RoboDK station: Proyecto_Grupo3_P105.rdk

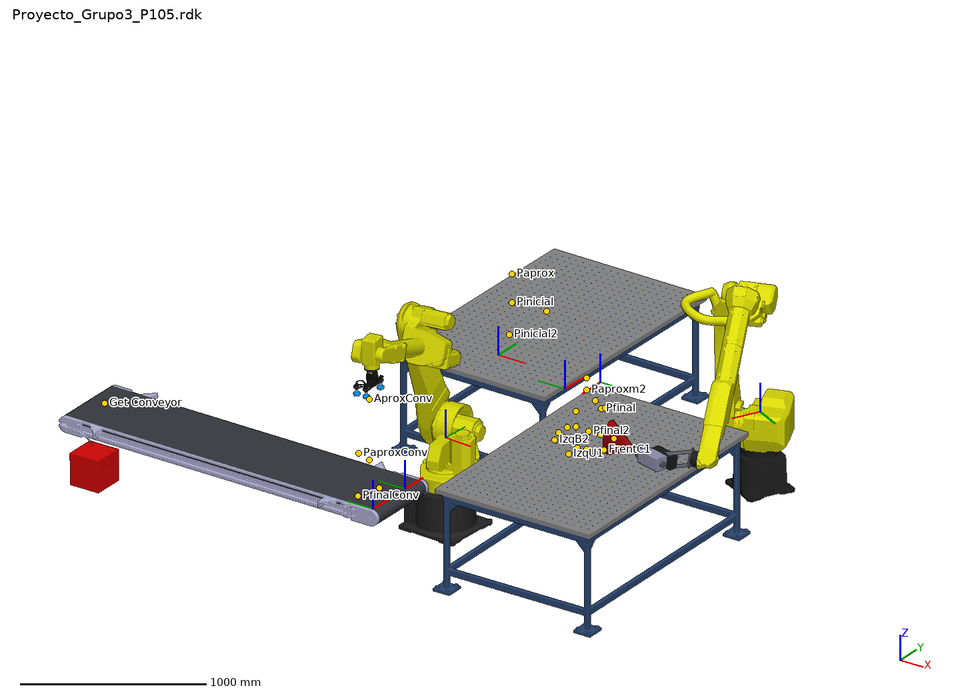
[picture v0: the station drawn from its stored meshes, robots at their saved joint values, targets as dots, program paths as lines]
Station ProyectoConConv (saved by RoboDK 5.3.0). Poses are relative to the parent item; angles as X-Y-Z fixed-axis rotations.
Station parameters (name, value as stored): ColorCilindro, 3.0
  - frame Fanuc M-16iB/20 Base at (-465.89, -504.82, 525) mm, rotated rx 0 ry 0 rz -2.81 deg
    - robot Fanuc M-16iB/20: 6 axes, payload 20 kg, reach 1667 mm, repeatability 0.08 mm, weight 270 kg
        modified DH rows (alpha deg, a mm, theta deg, d mm): 0, 0, 0, 525; -90, 150, -90, 0; 0, 770, 0, 0; -90, 100, 0, 740; 90, 0, 0, 0; -90, 0, 0, 100
        base shift (0, 0, -525) mm
        joint limits [-170, -90, -170, -200, -140, -450] to [170, 160, 290, 200, 140, 450]; home [0, 0, 0, 0, -90, 0]; saved at [100.119, -20.895, 160.194, 178.685, -110.161, -367.731]
      - tool RobotiQ EPick Four Vacuum Cup, TCP at (0, 21.99, 131.95) mm, size 175.2 x 107.7 x 135.6 mm
    - target Pfinal (Cartesian target) at (967.03, 121.53, 415.61) mm, rotated rx -178.82 ry 0.51 rz 89.06 deg; joints [7.493, 4.996, -18.964, 0.352, -72.278, -278.545] of Fanuc M-16iB/20
    - target PfinalConv (Cartesian target) at (196.13, -1019.55, 104.82) mm, rotated rx -178.83 ry 0.51 rz 177.59 deg; joints [-79.527, 21.76, -40.518, -0.315, -48.231, -102.682] of Fanuc M-16iB/20
    - target PaproxConv (Cartesian target) at (194.18, -1012.63, 357.54) mm, rotated rx -178.83 ry 0.51 rz 177.59 deg; joints [-79.563, 13.7, -22.039, -0.256, -66.709, -102.754] of Fanuc M-16iB/20
    - frame Est1 at (-300.91, 850, 79.96) mm, rotated rx 0 ry 0 rz 2.81 deg
      - target Paprox (Cartesian target) at (92.49, 0.53, 509.87) mm, rotated rx -178.82 ry 0.51 rz 89.06 deg; joints [105.312, -0.649, -5.743, 178.728, 84.484, -193.315] of Fanuc M-16iB/20
      - target Pinicial2 (Cartesian target) at (75, 0, 140) mm, rotated rx -180 ry 0.52 rz 90 deg; joints [-73.822, -24.597, 187.698, -180.122, -82.809, -13.348] of Fanuc M-16iB/20
      - target Pinicial (Cartesian target) at (93.45, -1.01, 339.4) mm, rotated rx -178.82 ry 0.51 rz 89.06 deg; joints [105.273, 0.25, -18.897, -1.336, -71.334, -372.97] of Fanuc M-16iB/20
      - target P2Inicial (Cartesian target) at (75, 350, 140) mm, rotated rx -178.82 ry 0.51 rz 90 deg; joints [102.152, 27.689, -21.607, -1.338, -68.714, -368.854] of Fanuc M-16iB/20
    - frame Est2 at (346.71, 909.84, 87.05) mm, rotated rx 0 ry 0 rz -86.3 deg
      - object Estacion2 at (1300, 499.97, 0) mm, rotated rx 0 ry 0 rz -180 deg, size 1535.8 x 1018.8 x 608.3 mm, geometry from Table-2000mmx1200mmx800mm.sld
      - target Paproxm2 (Cartesian target) at (800, 455.71, 400) mm, rotated rx 180 ry 0 rz 90 deg; joints [11.351, -2.011, -4.047, 0, -85.953, -367.648] of Fanuc M-16iB/20
      - target Pfinal2 (Cartesian target) at (775, 450, 140) mm, rotated rx -180 ry 0 rz 0 deg; joints [10.89, 2.514, -28.094, 0, -61.906, -97.187] of Fanuc M-16iB/20
      - object Estacion1 at (17.89, -650.14, -7.09) mm, rotated rx 0 ry 0 rz 179.11 deg, size 1535.8 x 1018.8 x 608.3 mm, geometry from Table-2000mmx1200mmx800mm.sld
  - Python program Set (listed below)
  - Python program Prepare (listed below)
  - Python program Robot1_2 (listed below)
  - Python program Robot2_Conv (listed below)
  - Python program Robot2_2 (listed below)
  - Python program SensorActivate (listed below)
  - frame Fanuc M-10iA/8L Base at (643.98, 857.38, 450) mm, rotated rx 0 ry 0 rz -116.36 deg
    - robot Fanuc M-10iA/8L: 6 axes, payload 8 kg, reach 2028 mm, repeatability 0.04 mm, weight 150 kg
        modified DH rows (alpha deg, a mm, theta deg, d mm): 0, 0, 0, 450; -90, 150, -90, 0; 0, 780, 0, 0; -90, 200, 0, 1080; 90, 0, 0, 0; -90, 0, 0, 100
        base shift (0, 0, -450) mm
        joint limits [-170, -90, -180, -200, -140, -270] to [170, 160, 267, 200, 140, 270]; home [12.06, 4.62, 10.35, -4.26, -75.46, -178.09]; saved at [47.67, 3.001, -39.586, 91.935, -94.481, -221.235]
      - tool Paint gun, TCP at (50, 0, 450) mm, rotated rx 0 ry 30 rz 0 deg, size 203.2 x 279.7 x 471.5 mm
    - target AproxPin (Cartesian target) at (1241.53, 330.16, 632.23) mm, rotated rx -179.35 ry -2.45 rz -157.72 deg; joints [13.753, -7.97, 9.222, -3.553, -71.889, -170.998] of Fanuc M-10iA/8L
    - target IzqU1 (Cartesian target) at (1385.42, 391.79, 236.72) mm, rotated rx 175.16 ry -45.65 rz -162.72 deg; joints [14.487, 30.06, -6.496, -3.483, -99.223, -180.287] of Fanuc M-10iA/8L
    - target IzqU2 (Cartesian target) at (1386.34, 378.43, 391.89) mm, rotated rx -176.7 ry -51.36 rz -166.63 deg; joints [15.972, 36.806, 3.248, 2.102, -114.653, -179.895] of Fanuc M-10iA/8L
    - target Sup1 (Cartesian target) at (1323.33, 361.68, 464.26) mm, rotated rx -179.35 ry -2.45 rz -157.72 deg; joints [14.303, -4.968, -0.111, -3.521, -62.54, -170.968] of Fanuc M-10iA/8L
    - target Sup2 (Cartesian target) at (1176.85, 310.11, 472.26) mm, rotated rx -178 ry 0.46 rz -156.27 deg; joints [13.626, -18.1, 1.596, -3.869, -61.306, -168.43] of Fanuc M-10iA/8L
    - target DerU1 (Cartesian target) at (1096.06, 271.61, 393.16) mm, rotated rx -177.41 ry 39.38 rz -154.65 deg; joints [7.092, -50.059, -3.563, -40.967, -22.985, -133.522] of Fanuc M-10iA/8L
    - target DerU2 (Cartesian target) at (1129.24, 280.47, 243.27) mm, rotated rx -176.98 ry 48.64 rz -154.02 deg; joints [6.444, -49.98, -15.791, -103.175, -16.992, -70.804] of Fanuc M-10iA/8L
    - target IzqB1 (Cartesian target) at (1352.99, 430.79, 281.25) mm, rotated rx 98.01 ry -2.72 rz -102.48 deg; joints [3.224, 45.691, -20.072, -62.199, -126.893, -145.453] of Fanuc M-10iA/8L
    - target IzqB2 (Cartesian target) at (1432.32, 316.89, 300.11) mm, rotated rx 98.01 ry -2.72 rz -102.48 deg; joints [-0.403, 53.002, -15.112, -63.442, -132.237, -149.123] of Fanuc M-10iA/8L
    - target AtrasB1 (Cartesian target) at (1371.24, 253.12, 300.21) mm, rotated rx 98.01 ry -2.72 rz -102.48 deg; joints [-2.438, 46.986, -18.398, -59.38, -132.376, -143.961] of Fanuc M-10iA/8L
    - target AtrasB2 (Cartesian target) at (1241.59, 206.8, 287.27) mm, rotated rx 98.01 ry -2.72 rz -102.48 deg; joints [-4.203, 36.509, -24.123, -53.707, -130.589, -136.372] of Fanuc M-10iA/8L
    - target IzqC1 (Cartesian target) at (1377.37, 326.06, 306.96) mm, rotated rx -88.88 ry 4.57 rz 171.9 deg; joints [-144.988, -47.039, 182.818, -87.325, -103.378, 174.474] of Fanuc M-10iA/8L
    - target IzqC2 (Cartesian target) at (1332.28, 498.61, 298.22) mm, rotated rx -90.14 ry 4.7 rz 156.34 deg; joints [-141.526, -71.736, 167.629, -79.805, -120.795, 191.683] of Fanuc M-10iA/8L
    - target FrentC1 (Cartesian target) at (1247.52, 535.75, 290.61) mm, rotated rx -87.43 ry 3.94 rz -168.8 deg; joints [-133.276, -36.716, 189.36, -86.769, -96.288, 168.888] of Fanuc M-10iA/8L
    - target FrentC2 (Cartesian target) at (1130.62, 430.13, 284.93) mm, rotated rx -87.14 ry 3.73 rz -164.4 deg; joints [-132.33, -23.306, 194.93, -86.372, -93.265, 163.449] of Fanuc M-10iA/8L
  - Python program pintura (listed below)
  - Python program SprayOn (listed below)
  - program MainProgram (15 instructions, listed below)
  - Python program Prog12 (listed below)
  - Python program PinturaP2 (listed below)
  - frame ConveyorReference at (-173.28, -1600, 618.68) mm, rotated rx 0 ry 0 rz 90.03 deg
    - target Get Conveyor (Cartesian target) at (200, 1900, 20) mm, rotated rx 90 ry 0 rz 0 deg; joints [0, 0, 0, 0, 0, 43.699]
    - frame Final_conv at (1800, 0, 0) mm
    - target Put Conveyor (Cartesian target) at (200, 100, 20) mm, rotated rx 90 ry 0 rz -180 deg; joints [134.006, 22.86, -66.558, 43.699, -45.994, 0]
    - object Conveyor at (0, 300, -50) mm, size 597 x 2090.8 x 107.2 mm
      - Python program RunConveyor (listed below)
      - Python program WaitForPart (listed below)
      - Python program SimulateGripper (listed below)
      - object box at (316.14, 335.9, 144.87) mm, rotated rx 0.06 ry -0.07 rz 75.08 deg, size 125 x 125 x 125 mm, geometry from box.sld
      - object Part 1 at (249.98, 1701.74, -449.97) mm, rotated rx 0.01 ry 1.18 rz 89.99 deg, size 187.5 x 187.5 x 187.5 mm, geometry from box.sld
      - object Part 2 at (250, 1704, -450) mm, rotated rx 0 ry 0 rz 90 deg, size 187.5 x 187.5 x 187.5 mm, geometry from box.sld
    - frame Inicial_conv at (300, 0, 0) mm
    - target FinalConv (Cartesian target) at (250, 200, 140) mm, rotated rx -178.82 ry 0.51 rz -180 deg; joints [100.119, -21.731, 187.781, 178.755, -82.581, -367.117] of Fanuc M-16iB/20
    - target AproxConv (Cartesian target) at (250, 200, 500) mm, rotated rx -178.82 ry 0.51 rz -180 deg; joints [100.119, -20.895, 160.194, 178.685, -110.161, -367.731] of Fanuc M-16iB/20

--- Python program Set ---
# Type help("robolink") or help("robodk") for more information
# Press F5 to run the script
# Note: you do not need to keep a copy of this file, your python script is saved with the station
from robolink import *    # API to communicate with RoboDK
from robodk import *      # basic matrix operations


#PARAM_SIZE_BOX = 'SizeBox'
#PARAM_SIZE_PALLET = 'SizePallet'
#PARAM_CONV_SPEED_MM = 'ConvSpeed'
PARAM_COLOR= 'ColorCilindro'



RDK = Robolink()

#size_box = RDK.getParam(PARAM_SIZE_BOX)
#size_pallet = RDK.getParam(PARAM_SIZE_PALLET)
#conv_speed = RDK.getParam(PARAM_CONV_SPEED_MM)
color = RDK.getParam(PARAM_COLOR)

# ------------------------------------------------------------
#size_box_input = mbox('Enter the size of the box in mm [L,W,H]', entry=size_box)
#if size_box_input:
#    RDK.setParam(PARAM_SIZE_BOX, size_box_input)
#else:
#    raise Exception('Operation cancelled by user')

# ------------------------------------------------------------
#size_pallet_input = mbox('Enter the size of the pallet', entry=size_pallet)
#if size_pallet_input:
#    RDK.setParam(PARAM_SIZE_PALLET, size_pallet_input)
#else:
#    raise Exception('Operation cancelled by user')

# ------------------------------------------------------------
#conv_speed_input = mbox('Enter the speed of the conveyor in mm/s', entry=conv_speed)
#if conv_speed_input:
#    RDK.setParam(PARAM_CONV_SPEED_MM, conv_speed_input)
#    conv_speed = float(conv_speed_input)
#    conv = RDK.Item('Conveyor Belt', ITEM_TYPE_ROBOT)
#    conv.setSpeed(conv_speed)

#else:
#    raise Exception('Operation cancelled by user')

# ------------------------------------------------------------
color_cilindro_input = mbox('Ingrese el color: 1:Amarillo 2:Azul 3:Rojo 4:Verde', entry=color)
if color_cilindro_input:
    RDK.setParam(PARAM_COLOR, color_cilindro_input)

else:
    raise Exception('Operation cancelled by user')

--- Python program Prepare ---
# Type help("robolink") or help("robodk") for more information
# Press F5 to run the script
# Note: you do not need to keep a copy of this file, your python script is saved with the station
from robolink import *    # API to communicate with RoboDK
from robodk import *      # basic matrix operations

# Use RoboDK API as RL
RDK = Robolink()

frame_pallet        = RDK.Item('Est1', ITEM_TYPE_FRAME)

# get variable parameters
#SIZE_BOX = RDK.getParam('SizeBox')
#SIZE_PALLET = RDK.getParam('SizePallet')
SIZE_BOX = [150,150,150]
SIZE_PALLET = [1,2,1]
#SIZE_BOX_XYZ = [float(x.replace(' ','')) for x in SIZE_BOX.split(',')]
#SIZE_PALLET_XYZ = [float(x.replace(' ','')) for x in SIZE_PALLET.split(',')]
SIZE_BOX_XYZ = [150,150,150]
SIZE_PALLET_XYZ = [1,2,1]
SIZE_BOX_Z = SIZE_BOX_XYZ[2] # the height of the boxes is important to take into account when approaching the positions

#COLOR_CILINDRO = RDK.getParam('ColorCilindro')
#COLOR_CILINDRO_RGB = [float(x.replace(' ','')) for x in COLOR_CILINDRO.split(',')]

def box_calc(size_xyz, pallet_xyz):
    """Calculates a list of points to store parts in a pallet"""
    [size_x, size_y, size_z] = size_xyz
    [pallet_x, pallet_y, pallet_z] = pallet_xyz
    xyz_list = []
    for h in range(int(pallet_z)):
        for j in range(int(pallet_y)):
            for i in range(int(pallet_x)):
                xyz_list = xyz_list + [[(i+0.5)*size_x, (j)*(size_y+200), (h+0)*size_z]]
    return xyz_list

def parts_setup(frame, positions, size_xyz):
    """Place a list of parts in a reference frame. The part/reference object must have been previously copied to the clipboard."""
    [size_x, size_y, size_z] = size_xyz
    nparts = len(positions)
    cstep = 1.0/(nparts - 1)
    for i in range(nparts):
        newpart = frame.Paste()
        newpart.Scale([(size_x/100), size_y/100, size_z/100]) #scale with respect to the reference object (100mm cube)
        newpart.setName('Part ' + str(i+1)) #set item name
        newpart.setPose(transl(positions[i])) #set item position with respect to parent
        newpart.setVisible(True, False) #make item visible but hide the reference frame
        newpart.Recolor([255/255,255/255,255/255,1]) #set RGBA color
#newpart.Recolor([1-cstep*i, cstep*i, 0.4, 1]) #set RGBA color

def cleanup(objects, startswith="Part "):
    """Deletes all objects where the name starts with "startswith", from the provided list of objects."""
    for item in objects:
        if item.Name().startswith(startswith):
            item.Delete()

# turn off rendering (much faster when setting up the station)
RDK.Render(False)

# cleanup previous simulation (generated parts and tools)
all_objects = RDK.ItemList(ITEM_TYPE_OBJECT, False)
cleanup(all_objects, 'Part ')
all_tools = RDK.ItemList(ITEM_TYPE_TOOL, False)
cleanup(all_tools, 'TCP ')

# copy the reference part
partref = RDK.Item('box')
partref.Copy()

#RL.Set_Simulation_Speed(500);
#RL.Set_Simulation_Mode(1)

# calculate an array of positions to get/store the parts
parts_positions = box_calc(SIZE_BOX_XYZ, SIZE_PALLET_XYZ)

# setup/initialise the parts on the palled
parts_setup(frame_pallet, parts_positions, SIZE_BOX_XYZ)

RDK.Render(True)

--- Python program Robot1_2 ---
# Type help("robolink") or help("robodk") for more information
# Press F5 to run the script
# Note: you do not need to keep a copy of this file, your python script is saved with the station
from robolink import *    # API to communicate with RoboDK
from robodk import *      # basic matrix operations

# Use RoboDK API as RL
RDK = Robolink()

# define default approach distance
APPROACH = 100

# gather robot, tool and reference frames from the station
robot = RDK.Item('Fanuc M-16iB/20', ITEM_TYPE_ROBOT)
tool = RDK.Item('RobotiQ EPick Four Vacuum Cup', ITEM_TYPE_TOOL)
frame_pallet = RDK.Item('Est1', ITEM_TYPE_FRAME)
frame_pallet2 = RDK.Item('Est2', ITEM_TYPE_FRAME)


# gather targets
target_aprox = RDK.Item('Paprox', ITEM_TYPE_TARGET)
target_aprox2 = RDK.Item('Paproxm2', ITEM_TYPE_TARGET)
target_final = RDK.Item('Pfinal2', ITEM_TYPE_TARGET)
target_inicial = RDK.Item('Pinicial2', ITEM_TYPE_TARGET)



def TCP_On(toolitem):
    """Attaches the closest object to the toolitem Htool pose,
    It will also output appropriate function calls on the generated robot program (call to TCP_On)"""
    toolitem.AttachClosest()
    toolitem.RDK().RunMessage('Set air valve on')
    toolitem.RDK().RunProgram('TCP_On()')

def TCP_Off(toolitem, itemleave=0):
    """Detaches the closest object attached to the toolitem Htool pose,
    It will also output appropriate function calls on the generated robot program (call to TCP_Off)"""
    toolitem.DetachAll(itemleave)
    toolitem.RDK().RunMessage('Set air valve off')
    toolitem.RDK().RunProgram('TCP_Off()')



# ---------------------------------------------------------------------------------
# -------------------------- PROGRAM START ----------------------------------------

tool_xyzrpw = tool.PoseTool()*transl(0,0,50)
tool_tcp = robot.AddTool(tool_xyzrpw, 'TCP A')

robot.setPoseTool(tool_tcp)
robot.setSpeed(100)
robot.setPoseFrame(frame_pallet)
robot.MoveJ(target_aprox)
#target_i_app = target_inicial * transl(0,0,-(APPROACH+50))
#robot.MoveJ(target_i_app)
#TCP_On(tool)
robot.MoveL(target_inicial)
robot.setSpeed(100)
TCP_On(tool)
#obj.setParentStatic(tool)
#TCP_On(tool)
#robot.MoveL(target_i_app)
robot.MoveL(target_aprox)
robot.setSpeed(100)
#TCP_On(tool)
robot.setPoseFrame(frame_pallet2)
robot.MoveL(target_aprox2)
robot.setSpeed(100)
robot.MoveL(target_final)
#robot.MoveJ(target_inicial)
TCP_Off(tool, frame_pallet2)
robot.MoveJ(target_aprox2)
robot.setPoseFrame(frame_pallet)
robot.MoveL(target_aprox)


def cleanup(objects, startswith="Part "):
    """Deletes all objects where the name starts with "startswith", from the provided list of objects."""
    for item in objects:
        if item.Name().startswith(startswith):
            item.Delete()

# turn off rendering (much faster when setting up the station)
RDK.Render(False)

# cleanup previous simulation (generated parts and tools)

all_tools = RDK.ItemList(ITEM_TYPE_TOOL, False)
cleanup(all_tools, 'TCP ')

--- Python program Robot2_Conv ---
# Type help("robolink") or help("robodk") for more information
# Press F5 to run the script
# Note: you do not need to keep a copy of this file, your python script is saved with the station
from robolink import *    # API to communicate with RoboDK
from robodk import *      # basic matrix operations

# Use RoboDK API as RL
RDK = Robolink()

# define default approach distance
#APPROACH = 100

# gather robot, tool and reference frames from the station
robot = RDK.Item('Fanuc M-16iB/20', ITEM_TYPE_ROBOT)
tool = RDK.Item('RobotiQ EPick Four Vacuum Cup', ITEM_TYPE_TOOL)
#obj = RDK.Item('box', ITEM_TYPE_OBJECT)
frame_pallet = RDK.Item('Est2', ITEM_TYPE_FRAME)
frame_pallet2 = RDK.Item('ConveyorReference', ITEM_TYPE_FRAME)
#frame_conv          = RDK.Item('ConveyorReference', ITEM_TYPE_FRAME)
#frame_conv_moving   = RDK.Item('MovingRef', ITEM_TYPE_FRAME)

# gather targets
target_aprox = RDK.Item('Paproxm2', ITEM_TYPE_TARGET)
target_aprox2 = RDK.Item('AproxConv', ITEM_TYPE_TARGET)
target_final = RDK.Item('FinalConv', ITEM_TYPE_TARGET)
target_inicial = RDK.Item('Pfinal2', ITEM_TYPE_TARGET)



def TCP_On(toolitem):
    """Attaches the closest object to the toolitem Htool pose,
    It will also output appropriate function calls on the generated robot program (call to TCP_On)"""
    toolitem.AttachClosest()
    toolitem.RDK().RunMessage('Set air valve on')
    toolitem.RDK().RunProgram('TCP_On()')

def TCP_Off(toolitem, itemleave=0):
    """Detaches the closest object attached to the toolitem Htool pose,
    It will also output appropriate function calls on the generated robot program (call to TCP_Off)"""
    toolitem.DetachAll(itemleave)
    toolitem.RDK().RunMessage('Set air valve off')
    toolitem.RDK().RunProgram('TCP_Off()')



# ---------------------------------------------------------------------------------
# -------------------------- PROGRAM START ----------------------------------------

tool_xyzrpw = tool.PoseTool()*transl(0,0,50)
tool_tcp = robot.AddTool(tool_xyzrpw, 'TCP B')

robot.setPoseTool(tool_tcp)

robot.setPoseFrame(frame_pallet)
robot.MoveJ(target_aprox)
TCP_On(tool)
robot.MoveJ(target_inicial)
#obj.setParentStatic(tool)
TCP_On(tool)
robot.MoveJ(target_aprox)
#TCP_On(tool)
robot.setPoseFrame(frame_pallet2)
robot.MoveL(target_aprox2)
robot.MoveL(target_final)
#robot.MoveJ(target_inicial)
TCP_Off(tool, frame_pallet2)
robot.MoveJ(target_aprox2)


def cleanup(objects, startswith="Part "):
    """Deletes all objects where the name starts with "startswith", from the provided list of objects."""
    for item in objects:
        if item.Name().startswith(startswith):
            item.Delete()

# turn off rendering (much faster when setting up the station)
RDK.Render(False)

# cleanup previous simulation (generated parts and tools)
all_tools = RDK.ItemList(ITEM_TYPE_TOOL, False)
cleanup(all_tools, 'TCP ')

--- Python program Robot2_2 ---
# Type help("robolink") or help("robodk") for more information
# Press F5 to run the script
# Note: you do not need to keep a copy of this file, your python script is saved with the station
from robolink import *    # API to communicate with RoboDK
from robodk import *      # basic matrix operations

# Use RoboDK API as RL
RDK = Robolink()

# define default approach distance
#APPROACH = 100

# gather robot, tool and reference frames from the station
robot = RDK.Item('Fanuc M-16iB/20', ITEM_TYPE_ROBOT)
tool = RDK.Item('RobotiQ EPick Four Vacuum Cup', ITEM_TYPE_TOOL)
#obj = RDK.Item('box', ITEM_TYPE_OBJECT)
frame_pallet = RDK.Item('Est1', ITEM_TYPE_FRAME)
frame_pallet2 = RDK.Item('Est2', ITEM_TYPE_FRAME)


# gather targets
target_aprox = RDK.Item('Paprox', ITEM_TYPE_TARGET)
target_aprox2 = RDK.Item('Paproxm2', ITEM_TYPE_TARGET)
target_final = RDK.Item('Pfinal2', ITEM_TYPE_TARGET)
target_inicial = RDK.Item('P2Inicial', ITEM_TYPE_TARGET)




def TCP_On(toolitem):
    """Attaches the closest object to the toolitem Htool pose,
    It will also output appropriate function calls on the generated robot program (call to TCP_On)"""
    toolitem.AttachClosest()
    toolitem.RDK().RunMessage('Set air valve on')
    toolitem.RDK().RunProgram('TCP_On()')

def TCP_Off(toolitem, itemleave=0):
    """Detaches the closest object attached to the toolitem Htool pose,
    It will also output appropriate function calls on the generated robot program (call to TCP_Off)"""
    toolitem.DetachAll(itemleave)
    toolitem.RDK().RunMessage('Set air valve off')
    toolitem.RDK().RunProgram('TCP_Off()')


# ---------------------------------------------------------------------------------
# -------------------------- PROGRAM START ----------------------------------------

tool_xyzrpw = tool.PoseTool()*transl(0,0,50)
tool_tcp = robot.AddTool(tool_xyzrpw, 'TCP C')

robot.setPoseTool(tool_tcp)

robot.setPoseFrame(frame_pallet)
robot.MoveJ(target_aprox)
TCP_On(tool)
robot.MoveL(target_inicial)
#obj.setParentStatic(tool)
TCP_On(tool)
robot.MoveJ(target_aprox)
#TCP_On(tool)
robot.setPoseFrame(frame_pallet2)
robot.MoveL(target_aprox2)
robot.MoveL(target_final)
#robot.MoveJ(target_inicial)
TCP_Off(tool, frame_pallet2)
robot.MoveJ(target_aprox2)
robot.setPoseFrame(frame_pallet)
robot.MoveL(target_aprox)


def cleanup(objects, startswith="Part "):
    """Deletes all objects where the name starts with "startswith", from the provided list of objects."""
    for item in objects:
        if item.Name().startswith(startswith):
            item.Delete()

# turn off rendering (much faster when setting up the station)
RDK.Render(False)

# cleanup previous simulation (generated parts and tools)

all_tools = RDK.ItemList(ITEM_TYPE_TOOL, False)
cleanup(all_tools, 'TCP ')

--- Python program SensorActivate ---
# Type help("robolink") or help("robodk") for more information
# Press F5 to run the script
# Note: you do not need to keep a copy of this file, your python script is saved with the station
from robolink import *    # API to communicate with RoboDK
from robodk import *      # basic matrix operations
RDK = Robolink()

# This script allows to simulate a laser sensor
# that detect the presence of a part in a plane,
# such as a part crossing a laser sensor in a
# conveyor belt

# Use a target from the station as a reference plane:
SENSOR_NAME = 'Sensor SICK WL4S'
SENSOR_VARIABLE = 'SENSOR'

# Look for parts with the keyword "Part"
PART_KEYWORD = 'Part '

# Update status every 1 ms
RECHECK_PERIOD = 0.001

# Get the sensor and the detection plane
SENSOR = RDK.Item(SENSOR_NAME, ITEM_TYPE_OBJECT)

# retrieve all objects
all_objects = RDK.ItemList(ITEM_TYPE_OBJECT, False)
part_objects = []
for obj in all_objects:
    if obj.Name().count(PART_KEYWORD) > 0:
        part_objects.append(obj)


# Loop forever to detect parts
detected_status = -1
while True:
    detected = 0
    for obj in part_objects:
        # check if an object has the part keyword and is detected by the laser
        if SENSOR.Collision(obj) > 0:
            detected = 1
            break

    # update the current status of the sensor
    if detected_status != detected:
        detected_status = detected
        RDK.setParam(SENSOR_VARIABLE, detected_status)
        print('Object detected status --> %i' % detected_status)

    # Wait some time...
    pause(RECHECK_PERIOD)

--- Python program pintura ---
#Type help("robolink") or help("robodk") for more information
# Press F5 to run the script
# Note: you do not need to keep a copy of this file, your python script is saved with the station
from robolink import *    # API to communicate with RoboDK
from robodk import *      # basic matrix operations

# Use RoboDK API as RL
RDK = Robolink()

# define default approach distance
#APPROACH = 100

# gather robot, tool and reference frames from the station
pieza= RDK.Item('Part 1', ITEM_TYPE_OBJECT)
pieza2= RDK.Item('Part 2', ITEM_TYPE_OBJECT)
robot = RDK.Item('Fanuc M-10iA/8L', ITEM_TYPE_ROBOT)
tool = RDK.Item('Paint gun', ITEM_TYPE_TOOL)

#frame_palletpin = RDK.Item('Frame 6', ITEM_TYPE_FRAME)
#frame_pallet2 = RDK.Item('Estacion2', ITEM_TYPE_FRAME)
COLOR_CILINDRO = RDK.getParam('ColorCilindro')
COLOR_CILINDRO_RGB = int(COLOR_CILINDRO)
ColorRGB=[]
if COLOR_CILINDRO_RGB == 1:  #Amarillo
    ColorRGB=[1,1,0,1]
if COLOR_CILINDRO_RGB == 2:  #Azul
    ColorRGB=[0,0,1,1]
if COLOR_CILINDRO_RGB == 3: #Rojo
    ColorRGB=[1,0,0,1]
if COLOR_CILINDRO_RGB == 4: #Verde
    ColorRGB=[0,128/255,0,1]

target_AproxPin = RDK.Item('AproxPin', ITEM_TYPE_TARGET)
target_IzqU1 = RDK.Item('IzqU1', ITEM_TYPE_TARGET)
target_IzqU2 = RDK.Item('IzqU2', ITEM_TYPE_TARGET)
target_Sup1 = RDK.Item('Sup1', ITEM_TYPE_TARGET)
target_Sup2 = RDK.Item('Sup2', ITEM_TYPE_TARGET)
target_DerU1 = RDK.Item('DerU1', ITEM_TYPE_TARGET)
target_DerU2 = RDK.Item('DerU2', ITEM_TYPE_TARGET)
target_IzqB1 = RDK.Item('IzqB1', ITEM_TYPE_TARGET)
target_IzqB2 = RDK.Item('IzqB2', ITEM_TYPE_TARGET)
target_AtrasB1 = RDK.Item('AtrasB1', ITEM_TYPE_TARGET)
target_AtrasB2 = RDK.Item('AtrasB2', ITEM_TYPE_TARGET)
target_IzqC1 = RDK.Item('IzqC1', ITEM_TYPE_TARGET)
target_IzqC2 = RDK.Item('IzqC2', ITEM_TYPE_TARGET)
target_FrentC1 = RDK.Item('FrentC1', ITEM_TYPE_TARGET)
target_FrentC2 = RDK.Item('FrentC2', ITEM_TYPE_TARGET)


#robot.setPoseFrame(frame_palletpin)
robot.MoveJ(target_AproxPin)
robot.MoveJ(target_IzqU1)
robot.MoveL(target_IzqU2)
robot.MoveL(target_Sup1)
robot.MoveL(target_Sup2)
robot.MoveL(target_DerU1)
robot.MoveL(target_DerU2)
robot.MoveJ(target_IzqB1)
robot.MoveL(target_IzqB2)
robot.MoveL(target_AtrasB1)
robot.MoveL(target_AtrasB2)
robot.MoveL(target_IzqC1)
robot.MoveL(target_IzqC2)
robot.MoveL(target_FrentC1)
robot.MoveL(target_FrentC2)

robot.setSpeed(100)
RDK.Spray_Clear()
pieza.Recolor(ColorRGB)
#pieza2.Recolor(ColorRGB)

--- Python program SprayOn ---
# This macro allows simulating a spray gun for painting or to simulate the trace of inspaction
#
# You can call SprayOn(1) to simulate turning the Spray gun ON or SprayOn(0) to stop simulating the gun
# Calling SprayOn(-1) clears all displayed data
# The macro will output spray gun statistics
#
# --------------------------------------------------------------
# This script shows how to create "spray" object in RoboDK that allows simulating particle deposition by using:
# RDK.Spray_Add(tool, object, options_command, volume, geometry)
#    tool: tool item (TCP) to use
#    object: object to project the particles
#    options_command (optional): string to specify options.
#    volume (optional): Matrix of parameters defining the volume of the spray gun
#    geometry (optional): Matrix of vertices defining the triangles.
#
# More information here:
# https://robodk.com/doc/en/PythonAPI/robolink.html#robolink.Robolink.Spray_Add
# https://robodk.com/doc/en/RoboDK-API.html
#
# The scripts ArcStart, ArcEnd and WeldOn and SpindleOn behave in a similar way, the only difference is the default behavior
# This behavior simmulates Fanuc Arc Welding and triggers appropriate output when using the customized post processor.
# Select ESC to clear the trace manually.
#
# Example scripts that use Spray_Add:
#     SpindleOn / SpindleOff    -> Turn trace On/Off
#     ArcOn / ArcOff            -> Turn trace On/Off
#     SprayOn / SprayOff        -> Simulate a spray given a workspace volume (for painting)
#     WeldOn / WeldOff          -> Support for multiple weld guns

#------------------------------------------------------------------

# Use a specific tool as a spray gun
Tool_Name = 'Paint gun'
#Tool_Name = 'Tool 2'

# Use a specific object to project particles:
Object_Name = 'Part 1'
#Object_Name = 'Part



# Define the default action (0 to deactivate, +1 to activate, -1 to clear any spray gun simulation)
# Setting it to None will display a message
ACTION = None

from robolink import *    # API to communicate with RoboDK
from robodk import *      # basic matrix operations
RDK = Robolink()

# quit if we are not in simulation mode
if RDK.RunMode() != RUNMODE_SIMULATE:
    quit()

# Get any previously added spray gun simulations and display statistics (spray on the part vs spray falling out of the part)
info, data = RDK.Spray_GetStats()
if data.size(1) > 0:
    print("Spray gun statistics:")
    print(info)
    print(data.tr())
    # # Diplay statistics
    # RDK.ShowMessage("Material used: %.1f%%<br>Material waisted: %.1f%%<br>Total particles: %.1f" % (data[1,0],data[2,0],data[3,0]), True)
    # # Clear previous spray
    # RDK.Spray_Clear()

# Check if we are running this program inside another program and passing arguments
import sys
if len(sys.argv) > 1:
    ACTION = int(sys.argv[1])

# If the default ACTION is None, display a message to activate/deactivate the spray gun
if ACTION is None:
    print('Note: This macro can be called as Spray(1) or SprayOn(0)')
    entry = mbox('Turn gun ON or OFF', ('On', '1'), ('Off', '0'))
    if not entry:
        quit()
    ACTION = int(entry)

if ACTION == 0:
    # Turn the gun off
    RDK.Spray_SetState(SPRAY_OFF)

elif ACTION < 0:
    # Clear all spray simulations (same as pressing ESC key)
    RDK.Spray_Clear()

elif ACTION > 0:
    # Create a new spray gun object in RoboDK
    # by using RDK.Spray_Add(tool, object, options_command, volume, geometry)
    # tool: tool item (TCP) to use
    # object: object to project the particles
    # options_command (optional): string to specify options. Example:
    #     STEP=AxB: Defines the grid to be projected 1x1 means only one line of particle projection (for example, for welding)
    #     PARTICLE: Defines the shape and size of particle (sphere or particle), unless a specific geometry is provided:
    #       a- SPHERE(radius, facets)
    #       b- SPHERE(radius, facets, scalex, scaley, scalez)
    #       b- CUBE(sizex, sizey, sizez)
    #     RAND=factor: Defines a random factor factor 0 means that the particles are not deposited randomly
    #     ELLYPSE: defines the volume as an ellypse (default)
    #     RECTANGLE: defines the volume as a rectangle
    #     PROJECT: project the particles to the surface (default) (for welding, painting or scanning)
    #     NO_PROJECT: does not project the particles to the surface (for example, for 3D printing)
    #
    # volume (optional): Matrix of parameters defining the volume of the spray gun
    # geometry (optional): Matrix of vertices defining the triangles.


    tool = 0    # auto detect active tool
    obj = 0     # auto detect object in active reference frame
    if Tool_Name is not None:
        tool = RDK.Item(Tool_Name, ITEM_TYPE_TOOL)

    if Object_Name is not None:
        obj = RDK.Item(Object_Name, ITEM_TYPE_OBJECT)
    # We can specify a given tool object and/or object
    #robot = RDK.Item("ABB IRB 2600-12/1.85", ITEM_TYPE_ROBOT)
    #tools = robot.Childs()
    #if len(tools) > 0:
    #    tool = tools[0]
    #obj = RDK.Item('object', ITEM_TYPE_OBJECT)

    #options_command = "ELLYPSE PROJECT PARTICLE=SPHERE(4,8,1,1,0.5) STEP=8x8 RAND=2" # simulate
    options_command = "PARTICLE=CUBE(10,10,2) STEP=8x8"
    #options_command = "PARTICLE=SPHERE(4,8) STEP=8x8"
    #options_command = "PARTICLE=SPHERE(4,8,1,1,0.1) STEP=8x8 RAND=3"

    # Example commands for welding:
    # options_command = "PROJECT PARTICLE=SPHERE(4,8)"
    # options_command = PARTICLE=SPHERE(4,8) STEP=1x0


    # define the ellypse volume as p0, pA, pB, colorRGBA (close and far), in mm
    # coordinates must be provided with respect to the TCP
    #close_p0 = [   -90,   -117, 0] # xyz in mm: Center of the conical ellypse (side 1)
    #close_pA = [   90,   -117, 0] # xyz in mm: First vertex of the conical ellypse (side 1)
    #close_pB = [   -90,  117, 0] # xyz in mm: Second vertex of the conical ellypse (side 1)
    #close_color = [ 1, 0, 0, 1]  # RGBA (0-1)

    #far_p0   = [   -175,   -190,  200] # xyz in mm: Center of the conical ellypse (side 2)
    #far_pA   = [  175,   -190,  200] # xyz in mm: First vertex of the conical ellypse (side 2)
    #far_pB   = [   -175, 190,  200] # xyz in mm: Second vertex of the conical ellypse (side 2)
    #far_color   = [ 0, 0, 1, 0.2]  # RGBA (0-1)

    #close_param = close_p0 + close_pA + close_pB + close_color
    #far_param = far_p0 + far_pA + far_pB + far_color
    #volume = Mat([close_param, far_param]).tr()
    #volume = Mat([close_param, far_param])
    #RDK.Spray_Add(tool, obj, options_command, volume.tr())
    #RDK.Spray_SetState(SPRAY_ON)
    COLOR_CILINDRO = RDK.getParam('ColorCilindro')
    COLOR_CILINDRO_RGB = int(COLOR_CILINDRO)
    ColorRGB=[]
    if COLOR_CILINDRO_RGB == 1:  #Amarillo
        ColorRGB=[1,1,0,1]
    if COLOR_CILINDRO_RGB == 2:  #Azul
        ColorRGB=[0,0,1,1]
    if COLOR_CILINDRO_RGB == 3: #Rojo
        ColorRGB=[1,0,0,1]
    if COLOR_CILINDRO_RGB == 4: #Verde
        ColorRGB=[0,128/255,0,1]

    # Another example with a varying rectancular shape
    # define the rectangular volume as p0, pA, pB, colorRGBA (close and far)
    close_param = [-90,-117,  0,  90,-117,0,   -90,117,  0,       ColorRGB[0],ColorRGB[1],ColorRGB[2],ColorRGB[3]]
    far_param   = [-175,-190,200, 175,-190,200,   -175,190,200,   ColorRGB[0],ColorRGB[1],ColorRGB[2],ColorRGB[3]]
    volume = Mat([close_param, far_param])
    RDK.Spray_Add(tool, obj, "RECTANGLE PARTICLE=SPHERE(2,5) STEP=15x15 RAND=3", volume.tr())
    RDK.Spray_SetState(SPRAY_ON)

    # Optional: define geometry as a list of triangles with normals (instead of a scaled cube or a sphere)
    # geom = Mat([[0,0,0,   0,0,1], [5,0,0,   0,0,1], [0,5,0,   0,0,1]])
    # RDK.Spray_Add(tool, obj, "STEP=8x8 RANDX=3", volume.tr(), geom.tr())
    # RDK.Spray_SetState(SPRAY_ON)

--- program MainProgram (robot Fanuc M-10iA/8L) ---
  Llamar Set
  Llamar Prepare
  Llamar Robot1_2
  Llamar SprayOn(1)
  Llamar pintura
  Llamar SprayOn(0)
  Llamar Robot2_Conv
  Ejecutar RunConveyor
  Llamar Set
  Llamar Robot2_2
  Llamar SprayOn(1)
  Llamar PinturaP2
  Llamar SprayOn(0)
  Llamar Robot2_Conv
  Ejecutar RunConveyor

--- Python program Prog12 ---
# Type help("robolink") or help("robodk") for more information
# Press F5 to run the script
# Note: you do not need to keep a copy of this file, your python script is saved with the station
from robolink import *    # API to communicate with RoboDK
from robodk import *      # basic matrix operations

# Use RoboDK API as RL
RDK = Robolink()

# define default approach distance
#APPROACH = 100

# gather robot, tool and reference frames from the station
robot = RDK.Item('Fanuc M-16iB/20', ITEM_TYPE_ROBOT)
tool = RDK.Item('RobotiQ EPick Four Vacuum Cup', ITEM_TYPE_TOOL)
#obj = RDK.Item('box', ITEM_TYPE_OBJECT)
frame_pallet = RDK.Item('Est2', ITEM_TYPE_FRAME)
frame_pallet2 = RDK.Item('Conveyor', ITEM_TYPE_FRAME)
#frame_conv          = RDK.Item('ConveyorReference', ITEM_TYPE_FRAME)
#frame_conv_moving   = RDK.Item('MovingRef', ITEM_TYPE_FRAME)

# gather targets
target_aprox = RDK.Item('Paproxm2', ITEM_TYPE_TARGET)
target_aprox2 = RDK.Item('AproxConv', ITEM_TYPE_TARGET)
target_final = RDK.Item('FinalConv', ITEM_TYPE_TARGET)
target_inicial = RDK.Item('Pfinal2', ITEM_TYPE_TARGET)



def TCP_On(toolitem):
    """Attaches the closest object to the toolitem Htool pose,
    It will also output appropriate function calls on the generated robot program (call to TCP_On)"""
    toolitem.AttachClosest()
    toolitem.RDK().RunMessage('Set air valve on')
    toolitem.RDK().RunProgram('TCP_On()')

def TCP_Off(toolitem, itemleave=0):
    """Detaches the closest object attached to the toolitem Htool pose,
    It will also output appropriate function calls on the generated robot program (call to TCP_Off)"""
    toolitem.DetachAll(itemleave)
    toolitem.RDK().RunMessage('Set air valve off')
    toolitem.RDK().RunProgram('TCP_Off()')

def WaitSensor():
    if RDK.RunMode() == RUNMODE_SIMULATE:
        # Simulate the sensor by waiting for the SENSOR status to turn to 1 (object present)
        while RDK.getParam(SENSOR_VARIABLE) == 0:
            pause(0.001)
    else:
        RDK.RunProgram('WaitSensor')
    print("Part detected")


# ---------------------------------------------------------------------------------
# -------------------------- PROGRAM START ----------------------------------------

tool_xyzrpw = tool.PoseTool()*transl(0,0,50)
tool_tcp = robot.AddTool(tool_xyzrpw, 'TCP D')

robot.setPoseTool(tool_tcp)

robot.setPoseFrame(frame_pallet2)
robot.MoveJ(target_aprox2)
WaitSensor()
robot.MoveL(target_inicial)
#obj.setParentStatic(tool)
TCP_On(tool)
robot.MoveJ(target_aprox)
#TCP_On(tool)
robot.setPoseFrame(frame_pallet2)
robot.MoveL(target_aprox2)
robot.MoveL(target_final)
#robot.MoveJ(target_inicial)
TCP_Off(tool, frame_pallet2)
robot.MoveJ(target_aprox2)


def cleanup(objects, startswith="Part "):
    """Deletes all objects where the name starts with "startswith", from the provided list of objects."""
    for item in objects:
        if item.Name().startswith(startswith):
            item.Delete()

# turn off rendering (much faster when setting up the station)
RDK.Render(False)

# cleanup previous simulation (generated parts and tools)
all_tools = RDK.ItemList(ITEM_TYPE_TOOL, False)
cleanup(all_tools, 'TCP ')







robot.setPoseTool(tool_tcp)
nparts = len(parts_positions)
i = 0
while i < nparts:
    # ----------- place the box i on the convegor ------
    # approach to the conveyor
    robot.setPoseFrame(frame_conv)
    target_conv_pose = target_conv.Pose()*transl(0,0,-SIZE_BOX_Z/2)
    target_conv_app = target_conv_pose*transl(0,0,-APPROACH)
    robot.MoveJ(target_conv_safe)
    robot.MoveJ(target_conv_app)
    WaitSensor()
    robot.MoveL(target_conv_pose)
    TCP_On(tool) # detach an place the object in the moving reference frame of the conveyor
    robot.MoveL(target_conv_app)
    robot.MoveJ(target_conv_safe)

    # ----------- take a part from the conveyor ------
    # get the xyz position of part i
    robot.setPose

--- Python program PinturaP2 ---
#Type help("robolink") or help("robodk") for more information
# Press F5 to run the script
# Note: you do not need to keep a copy of this file, your python script is saved with the station
from robolink import *    # API to communicate with RoboDK
from robodk import *      # basic matrix operations

# Use RoboDK API as RL
RDK = Robolink()

# define default approach distance
#APPROACH = 100

# gather robot, tool and reference frames from the station
pieza= RDK.Item('Part 1', ITEM_TYPE_OBJECT)
pieza2= RDK.Item('Part 2', ITEM_TYPE_OBJECT)
robot = RDK.Item('Fanuc M-10iA/8L', ITEM_TYPE_ROBOT)
tool = RDK.Item('Paint gun', ITEM_TYPE_TOOL)

frame_palletpin = RDK.Item('Frame 6', ITEM_TYPE_FRAME)
#frame_pallet2 = RDK.Item('Estacion2', ITEM_TYPE_FRAME)
COLOR_CILINDRO = RDK.getParam('ColorCilindro')
COLOR_CILINDRO_RGB = int(COLOR_CILINDRO)
ColorRGB=[]
if COLOR_CILINDRO_RGB == 1:  #Amarillo
    ColorRGB=[1,1,0,1]
if COLOR_CILINDRO_RGB == 2:  #Azul
    ColorRGB=[0,0,1,1]
if COLOR_CILINDRO_RGB == 3: #Rojo
    ColorRGB=[1,0,0,1]
if COLOR_CILINDRO_RGB == 4: #Verde
    ColorRGB=[0,128/255,0,1]

target_AproxPin = RDK.Item('AproxPin', ITEM_TYPE_TARGET)
target_IzqU1 = RDK.Item('IzqU1', ITEM_TYPE_TARGET)
target_IzqU2 = RDK.Item('IzqU2', ITEM_TYPE_TARGET)
target_Sup1 = RDK.Item('Sup1', ITEM_TYPE_TARGET)
target_Sup2 = RDK.Item('Sup2', ITEM_TYPE_TARGET)
target_DerU1 = RDK.Item('DerU1', ITEM_TYPE_TARGET)
target_DerU2 = RDK.Item('DerU2', ITEM_TYPE_TARGET)
target_IzqB1 = RDK.Item('IzqB1', ITEM_TYPE_TARGET)
target_IzqB2 = RDK.Item('IzqB2', ITEM_TYPE_TARGET)
target_AtrasB1 = RDK.Item('AtrasB1', ITEM_TYPE_TARGET)
target_AtrasB2 = RDK.Item('AtrasB2', ITEM_TYPE_TARGET)
target_IzqC1 = RDK.Item('IzqC1', ITEM_TYPE_TARGET)
target_IzqC2 = RDK.Item('IzqC2', ITEM_TYPE_TARGET)
target_FrentC1 = RDK.Item('FrentC1', ITEM_TYPE_TARGET)
target_FrentC2 = RDK.Item('FrentC2', ITEM_TYPE_TARGET)


#robot.setPoseFrame(frame_palletpin)
robot.MoveJ(target_AproxPin)
robot.MoveJ(target_IzqU1)
robot.MoveL(target_IzqU2)
robot.MoveL(target_Sup1)
robot.MoveL(target_Sup2)
robot.MoveL(target_DerU1)
robot.MoveL(target_DerU2)
robot.MoveJ(target_IzqB1)
robot.MoveL(target_IzqB2)
robot.MoveL(target_AtrasB1)
robot.MoveL(target_AtrasB2)
robot.MoveL(target_IzqC1)
robot.MoveL(target_IzqC2)
robot.MoveL(target_FrentC1)
robot.MoveL(target_FrentC2)

#robot.setSpeed(100)
RDK.Spray_Clear()
#pieza.Recolor(ColorRGB)
pieza2.Recolor(ColorRGB)

--- Python program RunConveyor ---
# Type help("robolink") or help("robodk") for more information
# Press F5 to run the script
# Note: you do not need to keep a copy of this file, your python script is saved with the station
from robolink import *    # API to communicate with RoboDK
from robodk import *      # basic matrix operations
RDK = Robolink()

# This script simulates a conveyor belt
CONVEYOR_NAME = 'Conveyor'
PICKABLE_OBJECTS_KEYWORD = 'Part'

# Speed of movement in MM/S with respect to the conveyor coordinates:
MOVE_SPEED_MMS = [0,20,0]
REFRESH_RATE = 0.005

# Define workspace of the conveyor to pick the objects:
CONV_SZ_X_MIN = 0
CONV_SZ_X_MAX = 440
CONV_SZ_Y_MIN = 0
CONV_SZ_Y_MAX = 2000
CONV_SZ_Z_MIN = -200
CONV_SZ_Z_MAX = +500

# Move objects that reached the end of the conveyor and were not picked:
FALLEN_OBJECTS = [0,0,-500]

# Get the conveyor item and reference for work space:
conv = RDK.Item(CONVEYOR_NAME)
conv_reference = conv.Parent()
poseconv = conv_reference.PoseAbs()

# One second in real life means 1 second of simulation. The simulation speed is taken from the station
SIMULATION_SPEED = 1

def is_inside_conveyor(pose):
    """Checks if a pose is inside the conveyor workspace"""
    pos = pose.Pos()
    if pos[0] > CONV_SZ_X_MIN and pos[0] < CONV_SZ_X_MAX and pos[1] > CONV_SZ_Y_MIN and pos[1] < CONV_SZ_Y_MAX and pos[2] > CONV_SZ_Z_MIN and pos[2] < CONV_SZ_Z_MAX:
        return True
    return False

def conveyor_move_object(pose, delta_time):
    """Moves the object pose through the conveyor depending on the time and speed"""
    delta_mm = mult3(MOVE_SPEED_MMS, delta_time)
    newpose = transl(delta_mm)*pose
    return newpose

# Get all objects (string list)
all_objects = RDK.ItemList(ITEM_TYPE_OBJECT, True)

# Convert object list into item pointers (faster)
# Also filter the list to take into account pickable objects only
objects = []
objects_name = []
objects_active = []
for i in range(len(all_objects)):
    if all_objects[i].count(PICKABLE_OBJECTS_KEYWORD) > 0:
        objects.append(RDK.Item(all_objects[i]))
        objects_name.append(all_objects[i])
        objects_active.append(False)

# The number of objects that can go in the conveyor
nobjects = len(objects)


# Infinite loop to simulate the conveyor behavior
current_time = 0
tic()
time_last = toc()
while True:
    # First: Look for objects that are not in the conveyor but are in the conveyor workspace
    for i in range(nobjects):
        obj_i = objects[i]

        # Skip if the object is already in the conveyor
        if objects_active[i]:
            continue

        # Check if the object has already been taken by a tool. If so, do not take it in the conveyor
        if obj_i.Parent().Type() == ITEM_TYPE_TOOL:
            continue

        # Check if the object is within the conveyor work area
        posei = obj_i.PoseAbs()
        poseirel = invH(poseconv)*posei
        if is_inside_conveyor(poseirel):
            # take the object
            obj_i.setParentStatic(conv)
            print('Adding object %s to the conveyor' % objects_name[i])
            objects_active[i] = True

    # Second step: Update the position of every object in the conveyor
    SIMULATION_SPEED = RDK.SimulationSpeed()
    time_current = toc()
    time_delta = time_current - time_last
    time_last = time_current
    current_time = current_time + time_delta*SIMULATION_SPEED

    # Make a list of objects with their matching positions to update
    obj_items = []
    obj_poses_abs = []
    for i in range(nobjects):
        obj_i = objects[i]

        # Check if the object has been picked from the conveyor
        if objects_active[i] and not obj_i.Parent().equals(conv):
            objects_active[i] = False
            print('Object %s was picked from the conveyor' % objects_name[i])
            continue

        # Skip update for objects that are not in the conveyor
        if not objects_active[i]:
            continue

        # Update the position of the object
        posei = invH(poseconv)*obj_i.PoseAbs()
        newposei = conveyor_move_object(posei, time_delta*SIMULATION_SPEED)
        if not is_inside_conveyor(newposei):
            print('Warning!! Object %s fell from the conveyor at %.1f seconds after simulation started' % (objects_name[i], current_time))
            #raise Exception('Object %s was not picked from the conveyor!' % objects_name[i])
            newposei = transl(FALLEN_OBJECTS)*newposei
            objects_active[i] = False

        #obj_i.setPose(newposei) # this will provoke a refresh (can be slow)
        obj_items.append(obj_i)
        obj_poses_abs.append(poseconv*newposei)

    # Update the object positions
    RDK.setPosesAbs(obj_items, obj_poses_abs)

    # Take a break...
    pause(REFRESH_RATE)

conv.Stop()

--- Python program WaitForPart ---
# Type help("robolink") or help("robodk") for more information
# Press F5 to run the script
# Note: you do not need to keep a copy of this file, your python script is saved with the station
from robolink import *    # API to communicate with RoboDK
from robodk import *      # basic matrix operations
RDK = Robolink()

# This script allows to simulate a laser sensor
# that detect the presence of a part in a plane,
# such as a part crossing a laser sensor in a
# conveyor belt

# The script finishes once a part has been detected
# so it works like a WAIT UNTIL function.

# Use a target from the station as a reference plane:
TARGET_NAME = 'Get Conveyor'
LASER_PLANE = [0,-1,0] # normal of the plane

# Activate within this tolerance
TOLERANCE_CHECK_MM = 10

# Look for parts with the keyword "Part"
PICKABLE_OBJECTS_KEYWORD = 'Part'

# Update status every 1 ms
RECHECK_PERIOD = 0.001

# Get the target and the detection plane
target = RDK.Item(TARGET_NAME)
targetpose = target.PoseAbs()
DETECT_PLANE_POINT = targetpose.Pos()
DETECT_PLANE_VECTOR = LASER_PLANE

# Define a function to detect a target
def part_detected(pos):
    """Check if a part is in the detection area (proximity of a point to a plane)"""
    pos_proj = proj_pt_2_plane(pos, DETECT_PLANE_POINT, DETECT_PLANE_VECTOR)
    distance2plane = norm(subs3(pos,pos_proj))
    if distance2plane < TOLERANCE_CHECK_MM:
        return True
    return False

# Get all object names
all_objects = RDK.ItemList(ITEM_TYPE_OBJECT, True)

# Get object items in a list (faster) and filter by keyword
check_objects = []
check_objects_names = []
for i in range(len(all_objects)):
    if all_objects[i].count(PICKABLE_OBJECTS_KEYWORD) > 0:
        check_objects_names.append(all_objects[i])
        check_objects.append(RDK.Item(all_objects[i]))

# Make sure that there are part that we are expecting
nCheck_objects = len(check_objects)
if nCheck_objects == 0:
    raise Exception('No parts to check for. The keyword is %s.' % PICKABLE_OBJECTS_KEYWORD)

# Loop forever until a part is detected by the sensor
part_available = False;
while not part_available:
    for i in range(nCheck_objects):
        if part_detected(check_objects[i].PoseAbs().Pos()):
            print('Part detected: %s' % check_objects_names[i])
            part_available = True
            break

    # Wait some time...
    pause(RECHECK_PERIOD)

print('Procedure finished')

--- Python program SimulateGripper ---
# Type help("robolink") or help("robodk") for more information
# Press F5 to run the script
# Note: you do not need to keep a copy of this file, your python script is saved with the station
from robolink import *    # API to communicate with RoboDK
from robodk import *      # basic matrix operations
RDK = Robolink()

# This file allows simulating the opening and closing of grippers.
# Two models of the gripper per robot are required: one opened and one closed.
# The opened model of the gripper should have the keyword "Opened"
# The closed model of the gripper should have the keyword "Closed"
# Simply place this file in the station and leave it running to
# make it work

OPENED_KEYWORD = 'Opened'
CLOSED_KEYWORD = 'Closed'
UPDATE_FREQUENCY = 0.01

# Loop forever
print('Starting infinite loop to simulate open/close of tools')
while True:
    # First step: get a list of tool pairs (open, closed) per robot
    Tool_Pairs = []
    # get all the robot names (strings)
    all_robots = RDK.ItemList(ITEM_TYPE_ROBOT)
    for i in range(len(all_robots)):
        roboti = RDK.Item(all_robots[i])
        roboti_name = roboti.Name()
        # get the tools of each robot
        roboti_tools = roboti.Childs()
        opened = None
        closed = None
        # store the opened model and closed model of each gripper
        for t in range(len(roboti_tools)):
            tnamei = roboti_tools[t].Name()
            if not isinstance(opened,Item) and tnamei.count(OPENED_KEYWORD) > 0:
                opened = roboti_tools[t]
                print('Using %s from robot %s as gripper opened' % (tnamei, roboti_name))
            elif not isinstance(closed,Item) and tnamei.count(CLOSED_KEYWORD) > 0:
                closed = roboti_tools[t]
                print('Using %s from robot %s as gripper closed' % (tnamei, roboti_name))

            if isinstance(opened, Item) and isinstance(closed, Item):
                # Stop if we have an open state and a closed state per robot
                break;
        Tool_Pairs.append([opened, closed])

    # We may find as many pairs of tools as robots are available in the station
    nTool_Pairs = len(Tool_Pairs)
    while True:
        #try:
            # Iterate through all tool pairs and detect the presence of objects
            for i in range(nTool_Pairs):
                opened = Tool_Pairs[i][0]
                closed = Tool_Pairs[i][1]
                open_valid = isinstance(opened,Item)
                close_valid = isinstance(closed,Item)
                tool_is_open = True

                # Check if the tool holds one or more objects:
                if (open_valid and len(opened.Childs()) > 0) or (close_valid and len(closed.Childs()) > 0):
                    tool_is_open = False

                # Update the visibility of the tools
                if open_valid:
                    opened.setVisible(tool_is_open)
                if close_valid:
                    closed.setVisible(not tool_is_open)

            # Take a pause...
            pause(UPDATE_FREQUENCY)

        #except:
            #print('An item was deleted. Remaking tool list')
            #break
